{attribute 'GeneratedUsingTerminal: EL6601--0000'}
{attribute addProperty BoxType "EL6601--0000"}
{attribute addProperty Id "EtcSlaveTerminalBaseInfoDataAT %I*InfoData_32EB74EA10"}
{attribute addProperty CRC "3667650902"}
{attribute addProperty Size "10"}
TYPE EL6601_DA9BE956 EXTENDS EtcSlaveTerminalBase :
STRUCT
	{attribute addProperty Name "InfoData"}
	InfoData : InfoData_32EB74EA;
END_STRUCT
END_TYPE

(* stored: Version 1.2.0.0, ProductVersion 3.1.4024.9
   DUT EL6601_DA9BE956: Id {f3c7ed1a-244b-4fdf-ae98-3ec6c47437b4} *)
